LIN {X 0,Y 104.793,Z 356.414,A -85,B 0,C 180,E1 -28295.245,E2 -28295.245} C_VEL
LIN {X 0,Y 103.647,Z 359.104,A -85,B 0,C 180,E1 -28297.183,E2 -28297.183} C_VEL
LIN {X 0,Y 96.406,Z 367.355,A -85,B 0,C 180,E1 -28301.678,E2 -28301.678} C_VEL
LIN {X 0,Y 90.767,Z 372.964,A -85,B 0,C 180,E1 -28305.825,E2 -28305.825} C_VEL
LIN {X 0,Y 84.492,Z 378.456,A -85,B 0,C 180,E1 -28311.403,E2 -28311.403} C_VEL
LIN {X 0,Y 79.25,Z 382.759,A -85,B 0,C 180,E1 -28317.854,E2 -28317.854} C_VEL
LIN {X 0,Y 76.317,Z 385.034,A -85,B 0,C 180,E1 -28322.584,E2 -28322.584} C_VEL
LIN {X 0,Y 73.868,Z 386.882,A -85,B 0,C 180,E1 -28327.631,E2 -28327.631} C_VEL
LIN {X 0,Y 72.01,Z 388.266,A -85,B 0,C 180,E1 -28332.975,E2 -28332.975} C_VEL
LIN {X 0,Y 70.538,Z 389.359,A -85,B 0,C 180,E1 -28339.552,E2 -28339.552} C_VEL
LIN {X 0,Y 69.778,Z 389.739,A -85,B 0,C 180,E1 -28342.701,E2 -28342.701} C_VEL
LIN {X 0,Y 68.056,Z 390.083,A -85,B 0,C 180,E1 -28347.417,E2 -28347.417} C_VEL
LIN {X 0,Y 64.284,Z 389.837,A -85,B 0,C 180,E1 -28359.106,E2 -28359.106} C_VEL
LIN {X 0,Y 64.171,Z 389.276,A -85,B 0,C 180,E1 -28364.414,E2 -28364.414} C_VEL
LIN {X 0,Y 64.494,Z 388.958,A -85,B 0,C 180,E1 -28366.15,E2 -28366.15} C_VEL
LIN {X 0,Y 67.351,Z 387.167,A -85,B 0,C 180,E1 -28374.671,E2 -28374.671} C_VEL
LIN {X 0,Y 71.592,Z 384.296,A -85,B 0,C 180,E1 -28382.679,E2 -28382.679} C_VEL
LIN {X 0,Y 76.945,Z 380.402,A -85,B 0,C 180,E1 -28389.746,E2 -28389.746} C_VEL
LIN {X 0,Y 83.424,Z 375.369,A -85,B 0,C 180,E1 -28395.733,E2 -28395.733} C_VEL
LIN {X 0,Y 90.542,Z 369.031,A -85,B 0,C 180,E1 -28400.916,E2 -28400.916} C_VEL
LIN {X 0,Y 98.216,Z 361.109,A -85,B 0,C 180,E1 -28405.373,E2 -28405.373} C_VEL
LIN {X 0,Y 99.699,Z 358.129,A -85,B 0,C 180,E1 -28407.77,E2 -28407.77} C_VEL
LIN {X 0,Y 100.292,Z 356.377,A -85,B 0,C 180,E1 -28409.361,E2 -28409.361} C_VEL
LIN {X 0,Y 100.745,Z 353.085,A -85,B 0,C 180,E1 -28413.037,E2 -28413.037} C_VEL
LIN {X 0,Y 100.845,Z 351.331,A -85,B 0,C 180,E1 -28415.282,E2 -28415.282} C_VEL
LIN {X 0,Y 100.69,Z 348.475,A -85,B 0,C 180,E1 -28419.574,E2 -28419.574} C_VEL
LIN {X 0,Y 100.47,Z 346.218,A -85,B 0,C 180,E1 -28423.751,E2 -28423.751} C_VEL
LIN {X 0,Y 100.246,Z 344.108,A -85,B 0,C 180,E1 -28428.967,E2 -28428.967} C_VEL
LIN {X 0,Y 100.132,Z 342.512,A -85,B 0,C 180,E1 -28435.975,E2 -28435.975} C_VEL
LIN {X 0,Y 100.538,Z 341.834,A -85,B 0,C 180,E1 -28440,E2 -28440} C_VEL
LIN {X 0,Y 100.479,Z 343.621,A -85,B 0,C 180,E1 -28448.041,E2 -28448.041} C_VEL
LIN {X 0,Y 100.756,Z 345.239,A -85,B 0,C 180,E1 -28452.434,E2 -28452.434} C_VEL
LIN {X 0,Y 100.752,Z 348.841,A -85,B 0,C 180,E1 -28458.294,E2 -28458.294} C_VEL
LIN {X 0,Y 100.473,Z 352.18,A -85,B 0,C 180,E1 -28462.454,E2 -28462.454} C_VEL
LIN {X 0,Y 99.589,Z 357.923,A -85,B 0,C 180,E1 -28468.447,E2 -28468.447} C_VEL
LIN {X 0,Y 99.259,Z 359.239,A -85,B 0,C 180,E1 -28469.711,E2 -28469.711} C_VEL
LIN {X 0,Y 95.481,Z 365.627,A -85,B 0,C 180,E1 -28474.098,E2 -28474.098} C_VEL
LIN {X 0,Y 94.457,Z 367.013,A -85,B 0,C 180,E1 -28475.07,E2 -28475.07} C_VEL
LIN {X 0,Y 86.861,Z 374.432,A -85,B 0,C 180,E1 -28479.766,E2 -28479.766} C_VEL
LIN {X 0,Y 80.095,Z 380.399,A -85,B 0,C 180,E1 -28485.414,E2 -28485.414} C_VEL
LIN {X 0,Y 73.98,Z 385.109,A -85,B 0,C 180,E1 -28491.866,E2 -28491.866} C_VEL
LIN {X 0,Y 68.92,Z 388.71,A -85,B 0,C 180,E1 -28499.344,E2 -28499.344} C_VEL
LIN {X 0,Y 66.352,Z 390.571,A -85,B 0,C 180,E1 -28504.932,E2 -28504.932} C_VEL
LIN {X 0,Y 64.453,Z 391.97,A -85,B 0,C 180,E1 -28510.905,E2 -28510.905} C_VEL
LIN {X 0,Y 63.178,Z 392.971,A -85,B 0,C 180,E1 -28517.144,E2 -28517.144} C_VEL
LIN {X 0,Y 62.555,Z 393.585,A -85,B 0,C 180,E1 -28523.549,E2 -28523.549} C_VEL
LIN {X 0,Y 62.607,Z 393.802,A -85,B 0,C 180,E1 -28529.999,E2 -28529.999} C_VEL
LIN {X 0,Y 62.554,Z 393.565,A -85,B 0,C 180,E1 -28536.45,E2 -28536.45} C_VEL
LIN {X 0,Y 63.173,Z 392.94,A -85,B 0,C 180,E1 -28542.855,E2 -28542.855} C_VEL
LIN {X 0,Y 64.448,Z 391.926,A -85,B 0,C 180,E1 -28549.095,E2 -28549.095} C_VEL
LIN {X 0,Y 66.351,Z 390.508,A -85,B 0,C 180,E1 -28555.067,E2 -28555.067} C_VEL
LIN {X 0,Y 70.489,Z 387.549,A -85,B 0,C 180,E1 -28563.255,E2 -28563.255} C_VEL
LIN {X 0,Y 75.858,Z 383.553,A -85,B 0,C 180,E1 -28570.43,E2 -28570.43} C_VEL
LIN {X 0,Y 82.788,Z 377.962,A -85,B 0,C 180,E1 -28576.999,E2 -28576.999} C_VEL
LIN {X 0,Y 90.604,Z 370.717,A -85,B 0,C 180,E1 -28582.662,E2 -28582.662} C_VEL
LIN {X 0,Y 94.437,Z 366.784,A -85,B 0,C 180,E1 -28584.946,E2 -28584.946} C_VEL
LIN {X 0,Y 98.282,Z 360.732,A -85,B 0,C 180,E1 -28589.104,E2 -28589.104} C_VEL
LIN {X 0,Y 99.138,Z 359.09,A -85,B 0,C 180,E1 -28590.249,E2 -28590.249} C_VEL
LIN {X 0,Y 100.072,Z 354.239,A -85,B 0,C 180,E1 -28595.079,E2 -28595.079} C_VEL
LIN {X 0,Y 100.485,Z 350.318,A -85,B 0,C 180,E1 -28599.531,E2 -28599.531} C_VEL
LIN {X 0,Y 100.597,Z 347.225,A -85,B 0,C 180,E1 -28603.773,E2 -28603.773} C_VEL
LIN {X 0,Y 100.675,Z 345.864,A -85,B 0,C 180,E1 -28605.858,E2 -28605.858} C_VEL
LIN {X 0,Y 100.584,Z 344.822,A -85,B 0,C 180,E1 -28608.014,E2 -28608.014} C_VEL
LIN {X 0,Y 100.327,Z 343.386,A -85,B 0,C 180,E1 -28611.946,E2 -28611.946} C_VEL
LIN {X 0,Y 100.495,Z 341.438,A -85,B 0,C 180,E1 -28620,E2 -28620} C_VEL
LIN {X 0,Y 100.058,Z 343.703,A -85,B 0,C 180,E1 -28630.472,E2 -28630.472} C_VEL
LIN {X 0,Y 100.312,Z 345.977,A -85,B 0,C 180,E1 -28636.275,E2 -28636.275} C_VEL
LIN {X 0,Y 100.573,Z 349.257,A -85,B 0,C 180,E1 -28642.047,E2 -28642.047} C_VEL
LIN {X 0,Y 100.754,Z 351.181,A -85,B 0,C 180,E1 -28644.933,E2 -28644.933} C_VEL
LIN {X 0,Y 100.621,Z 353.725,A -85,B 0,C 180,E1 -28648.128,E2 -28648.128} C_VEL
LIN {X 0,Y 100.212,Z 356.032,A -85,B 0,C 180,E1 -28650.563,E2 -28650.563} C_VEL
LIN {X 0,Y 99.055,Z 359.33,A -85,B 0,C 180,E1 -28653.525,E2 -28653.525} C_VEL
LIN {X 0,Y 98.237,Z 360.784,A -85,B 0,C 180,E1 -28654.645,E2 -28654.645} C_VEL
LIN {X 0,Y 90.606,Z 368.761,A -85,B 0,C 180,E1 -28659.135,E2 -28659.135} C_VEL
LIN {X 0,Y 83.478,Z 375.163,A -85,B 0,C 180,E1 -28664.307,E2 -28664.307} C_VEL
LIN {X 0,Y 76.994,Z 380.242,A -85,B 0,C 180,E1 -28670.286,E2 -28670.286} C_VEL
LIN {X 0,Y 71.622,Z 384.178,A -85,B 0,C 180,E1 -28677.338,E2 -28677.338} C_VEL
LIN {X 0,Y 67.358,Z 387.082,A -85,B 0,C 180,E1 -28685.333,E2 -28685.333} C_VEL
LIN {X 0,Y 65.247,Z 388.467,A -85,B 0,C 180,E1 -28691.148,E2 -28691.148} C_VEL
LIN {X 0,Y 62.941,Z 390.052,A -85,B 0,C 180,E1 -28703.59,E2 -28703.59} C_VEL
LIN {X 0,Y 62.722,Z 390.274,A -85,B 0,C 180,E1 -28710.001,E2 -28710.001} C_VEL
LIN {X 0,Y 62.941,Z 390.078,A -85,B 0,C 180,E1 -28716.412,E2 -28716.412} C_VEL
LIN {X 0,Y 64.494,Z 388.958,A -85,B 0,C 180,E1 -28726.15,E2 -28726.15} C_VEL
LIN {X 0,Y 65.325,Z 388.093,A -85,B 0,C 180,E1 -28731.256,E2 -28731.256} C_VEL
LIN {X 0,Y 65.947,Z 386.149,A -85,B 0,C 180,E1 -28739.749,E2 -28739.749} C_VEL
LIN {X 0,Y 67.198,Z 384.11,A -85,B 0,C 180,E1 -28746.298,E2 -28746.298} C_VEL
LIN {X 0,Y 69.308,Z 382.218,A -85,B 0,C 180,E1 -28750.671,E2 -28750.671} C_VEL
LIN {X 0,Y 70.305,Z 381.487,A -85,B 0,C 180,E1 -28751.943,E2 -28751.943} C_VEL
LIN {X 0,Y 78.633,Z 375.567,A -85,B 0,C 180,E1 -28759.439,E2 -28759.439} C_VEL
LIN {X 0,Y 86.244,Z 369.229,A -85,B 0,C 180,E1 -28764.579,E2 -28764.579} C_VEL
LIN {X 0,Y 93.006,Z 362.777,A -85,B 0,C 180,E1 -28768.22,E2 -28768.22} C_VEL
LIN {X 0,Y 93.91,Z 361.331,A -85,B 0,C 180,E1 -28769.385,E2 -28769.385} C_VEL
LIN {X 0,Y 94.71,Z 359.575,A -85,B 0,C 180,E1 -28771.164,E2 -28771.164} C_VEL
LIN {X 0,Y 95.354,Z 356.566,A -85,B 0,C 180,E1 -28774.987,E2 -28774.987} C_VEL
LIN {X 0,Y 95.522,Z 354.36,A -85,B 0,C 180,E1 -28778.415,E2 -28778.415} C_VEL
LIN {X 0,Y 95.604,Z 351.962,A -85,B 0,C 180,E1 -28782.899,E2 -28782.899} C_VEL
LIN {X 0,Y 95.525,Z 350.184,A -85,B 0,C 180,E1 -28787.249,E2 -28787.249} C_VEL
LIN {X 0,Y 95.559,Z 348.88,A -85,B 0,C 180,E1 -28791.541,E2 -28791.541} C_VEL
LIN {X 0,Y 96.103,Z 347.425,A -85,B 0,C 180,E1 -28800,E2 -28800} C_VEL
LIN {X 0,Y 95.893,Z 349.285,A -85,B 0,C 180,E1 -28808.429,E2 -28808.429} C_VEL
LIN {X 0,Y 95.97,Z 350.846,A -85,B 0,C 180,E1 -28812.691,E2 -28812.691} C_VEL
LIN {X 0,Y 95.697,Z 353.545,A -85,B 0,C 180,E1 -28817.306,E2 -28817.306} C_VEL
LIN {X 0,Y 94.847,Z 357.84,A -85,B 0,C 180,E1 -28822.935,E2 -28822.935} C_VEL
LIN {X 0,Y 93.979,Z 361.101,A -85,B 0,C 180,E1 -28826.66,E2 -28826.66} C_VEL
LIN {X 0,Y 93.253,Z 362.663,A -85,B 0,C 180,E1 -28828.099,E2 -28828.099} C_VEL
LIN {X 0,Y 90.33,Z 366.803,A -85,B 0,C 180,E1 -28831.147,E2 -28831.147} C_VEL
LIN {X 0,Y 89.184,Z 368.175,A -85,B 0,C 180,E1 -28832.097,E2 -28832.097} C_VEL
LIN {X 0,Y 81.199,Z 375.347,A -85,B 0,C 180,E1 -28836.81,E2 -28836.81} C_VEL
LIN {X 0,Y 72.857,Z 381.889,A -85,B 0,C 180,E1 -28843.657,E2 -28843.657} C_VEL
LIN {X 0,Y 66.526,Z 386.217,A -85,B 0,C 180,E1 -28850.664,E2 -28850.664} C_VEL
LIN {X 0,Y 62.902,Z 388.511,A -85,B 0,C 180,E1 -28856.037,E2 -28856.037} C_VEL
LIN {X 0,Y 59.955,Z 390.37,A -85,B 0,C 180,E1 -28862.037,E2 -28862.037} C_VEL
LIN {X 0,Y 57.762,Z 391.77,A -85,B 0,C 180,E1 -28868.591,E2 -28868.591} C_VEL
LIN {X 0,Y 56.266,Z 392.772,A -85,B 0,C 180,E1 -28875.533,E2 -28875.533} C_VEL
LIN {X 0,Y 55.513,Z 393.385,A -85,B 0,C 180,E1 -28882.726,E2 -28882.726} C_VEL
LIN {X 0,Y 55.506,Z 393.602,A -85,B 0,C 180,E1 -28889.999,E2 -28889.999} C_VEL
LIN {X 0,Y 55.511,Z 393.366,A -85,B 0,C 180,E1 -28897.273,E2 -28897.273} C_VEL
LIN {X 0,Y 56.262,Z 392.74,A -85,B 0,C 180,E1 -28904.467,E2 -28904.467} C_VEL
LIN {X 0,Y 57.758,Z 391.725,A -85,B 0,C 180,E1 -28911.409,E2 -28911.409} C_VEL
LIN {X 0,Y 59.954,Z 390.306,A -85,B 0,C 180,E1 -28917.962,E2 -28917.962} C_VEL
LIN {X 0,Y 64.658,Z 387.348,A -85,B 0,C 180,E1 -28926.714,E2 -28926.714} C_VEL
LIN {X 0,Y 70.589,Z 383.351,A -85,B 0,C 180,E1 -28934.181,E2 -28934.181} C_VEL
LIN {X 0,Y 77.441,Z 378.285,A -85,B 0,C 180,E1 -28940.333,E2 -28940.333} C_VEL
LIN {X 0,Y 85.131,Z 371.751,A -85,B 0,C 180,E1 -28945.644,E2 -28945.644} C_VEL
LIN {X 0,Y 89.174,Z 367.943,A -85,B 0,C 180,E1 -28947.911,E2 -28947.911} C_VEL
LIN {X 0,Y 93.145,Z 362.521,A -85,B 0,C 180,E1 -28951.848,E2 -28951.848} C_VEL
LIN {X 0,Y 93.986,Z 360.476,A -85,B 0,C 180,E1 -28953.808,E2 -28953.808} C_VEL
LIN {X 0,Y 94.958,Z 356.609,A -85,B 0,C 180,E1 -28958.281,E2 -28958.281} C_VEL
LIN {X 0,Y 95.591,Z 353.198,A -85,B 0,C 180,E1 -28962.897,E2 -28962.897} C_VEL
LIN {X 0,Y 95.85,Z 350.624,A -85,B 0,C 180,E1 -28967.293,E2 -28967.293} C_VEL
LIN {X 0,Y 95.769,Z 349.057,A -85,B 0,C 180,E1 -28971.56,E2 -28971.56} C_VEL
LIN {X 0,Y 96.064,Z 347.06,A -85,B 0,C 180,E1 -28980,E2 -28980} C_VEL
LIN {X 0,Y 95.417,Z 348.65,A -85,B 0,C 180,E1 -28988.471,E2 -28988.471} C_VEL
LIN {X 0,Y 95.402,Z 349.929,A -85,B 0,C 180,E1 -28992.768,E2 -28992.768} C_VEL
LIN {X 0,Y 95.48,Z 351.717,A -85,B 0,C 180,E1 -28997.123,E2 -28997.123} C_VEL
LIN {X 0,Y 95.418,Z 355.078,A -85,B 0,C 180,E1 -29003.236,E2 -29003.236} C_VEL
LIN {X 0,Y 94.965,Z 358.049,A -85,B 0,C 180,E1 -29007.368,E2 -29007.368} C_VEL
LIN {X 0,Y 93.898,Z 361.013,A -85,B 0,C 180,E1 -29010.605,E2 -29010.605} C_VEL
LIN {X 0,Y 93.003,Z 362.465,A -85,B 0,C 180,E1 -29011.778,E2 -29011.778} C_VEL
LIN {X 0,Y 85.01,Z 370.125,A -85,B 0,C 180,E1 -29016.288,E2 -29016.288} C_VEL
LIN {X 0,Y 76.266,Z 377.17,A -85,B 0,C 180,E1 -29022.506,E2 -29022.506} C_VEL
LIN {X 0,Y 69.596,Z 381.857,A -85,B 0,C 180,E1 -29028.975,E2 -29028.975} C_VEL
LIN {X 0,Y 64.014,Z 385.437,A -85,B 0,C 180,E1 -29036.706,E2 -29036.706} C_VEL
LIN {X 0,Y 60.985,Z 387.283,A -85,B 0,C 180,E1 -29042.551,E2 -29042.551} C_VEL
LIN {X 0,Y 58.577,Z 388.667,A -85,B 0,C 180,E1 -29048.904,E2 -29048.904} C_VEL
LIN {X 0,Y 55.909,Z 390.252,A -85,B 0,C 180,E1 -29062.779,E2 -29062.779} C_VEL
LIN {X 0,Y 55.649,Z 390.474,A -85,B 0,C 180,E1 -29070.001,E2 -29070.001} C_VEL
LIN {X 0,Y 55.909,Z 390.277,A -85,B 0,C 180,E1 -29077.222,E2 -29077.222} C_VEL
LIN {X 0,Y 58.576,Z 388.725,A -85,B 0,C 180,E1 -29091.098,E2 -29091.098} C_VEL
LIN {X 0,Y 60.977,Z 387.366,A -85,B 0,C 180,E1 -29097.454,E2 -29097.454} C_VEL
LIN {X 0,Y 65.724,Z 384.495,A -85,B 0,C 180,E1 -29106.025,E2 -29106.025} C_VEL
LIN {X 0,Y 70.305,Z 381.487,A -85,B 0,C 180,E1 -29111.943,E2 -29111.943} C_VEL
LIN {X 0,Y 73.125,Z 379.246,A -85,B 0,C 180,E1 -29115.692,E2 -29115.692} C_VEL
LIN {X 0,Y 76.946,Z 375.192,A -85,B 0,C 180,E1 -29121.978,E2 -29121.978} C_VEL
LIN {X 0,Y 81.339,Z 370.522,A -85,B 0,C 180,E1 -29127.46,E2 -29127.46} C_VEL
LIN {X 0,Y 84.847,Z 367.257,A -85,B 0,C 180,E1 -29129.866,E2 -29129.866} C_VEL
LIN {X 0,Y 88.03,Z 364.33,A -85,B 0,C 180,E1 -29131.428,E2 -29131.428} C_VEL
LIN {X 0,Y 88.837,Z 363.193,A -85,B 0,C 180,E1 -29132.531,E2 -29132.531} C_VEL
LIN {X 0,Y 89.409,Z 361.74,A -85,B 0,C 180,E1 -29134.408,E2 -29134.408} C_VEL
LIN {X 0,Y 89.91,Z 360.045,A -85,B 0,C 180,E1 -29136.993,E2 -29136.993} C_VEL
LIN {X 0,Y 90.324,Z 357.435,A -85,B 0,C 180,E1 -29141.866,E2 -29141.866} C_VEL
LIN {X 0,Y 90.45,Z 355.628,A -85,B 0,C 180,E1 -29146.52,E2 -29146.52} C_VEL
LIN {X 0,Y 90.604,Z 354.253,A -85,B 0,C 180,E1 -29151.075,E2 -29151.075} C_VEL
LIN {X 0,Y 91.347,Z 352.774,A -85,B 0,C 180,E1 -29160,E2 -29160} C_VEL
LIN {X 0,Y 91.033,Z 353.566,A -85,B 0,C 180,E1 -29164.428,E2 -29164.428} C_VEL
LIN {X 0,Y 90.954,Z 354.674,A -85,B 0,C 180,E1 -29168.89,E2 -29168.89} C_VEL
LIN {X 0,Y 90.738,Z 356.498,A -85,B 0,C 180,E1 -29173.436,E2 -29173.436} C_VEL
LIN {X 0,Y 90.028,Z 359.286,A -85,B 0,C 180,E1 -29178.195,E2 -29178.195} C_VEL
LIN {X 0,Y 88.752,Z 363.063,A -85,B 0,C 180,E1 -29183.324,E2 -29183.324} C_VEL
LIN {X 0,Y 88.142,Z 364.523,A -85,B 0,C 180,E1 -29185.06,E2 -29185.06} C_VEL
LIN {X 0,Y 85.452,Z 367.967,A -85,B 0,C 180,E1 -29187.853,E2 -29187.853} C_VEL
LIN {X 0,Y 82.726,Z 370.525,A -85,B 0,C 180,E1 -29189.448,E2 -29189.448} C_VEL
LIN {X 0,Y 75.787,Z 376.169,A -85,B 0,C 180,E1 -29193.424,E2 -29193.424} C_VEL
LIN {X 0,Y 68.138,Z 381.69,A -85,B 0,C 180,E1 -29199.323,E2 -29199.323} C_VEL
LIN {X 0,Y 61.187,Z 386.018,A -85,B 0,C 180,E1 -29206.435,E2 -29206.435} C_VEL
LIN {X 0,Y 57.141,Z 388.311,A -85,B 0,C 180,E1 -29212.049,E2 -29212.049} C_VEL
LIN {X 0,Y 53.751,Z 390.17,A -85,B 0,C 180,E1 -29218.465,E2 -29218.465} C_VEL
LIN {X 0,Y 51.175,Z 391.569,A -85,B 0,C 180,E1 -29225.669,E2 -29225.669} C_VEL
LIN {X 0,Y 48.473,Z 393.185,A -85,B 0,C 180,E1 -29241.663,E2 -29241.663} C_VEL
LIN {X 0,Y 48.423,Z 393.403,A -85,B 0,C 180,E1 -29249.999,E2 -29249.999} C_VEL
LIN {X 0,Y 48.472,Z 393.165,A -85,B 0,C 180,E1 -29258.336,E2 -29258.336} C_VEL
LIN {X 0,Y 51.171,Z 391.524,A -85,B 0,C 180,E1 -29274.332,E2 -29274.332} C_VEL
LIN {X 0,Y 53.749,Z 390.104,A -85,B 0,C 180,E1 -29281.535,E2 -29281.535} C_VEL
LIN {X 0,Y 59.088,Z 387.146,A -85,B 0,C 180,E1 -29290.856,E2 -29290.856} C_VEL
LIN {X 0,Y 65.674,Z 383.15,A -85,B 0,C 180,E1 -29298.511,E2 -29298.511} C_VEL
LIN {X 0,Y 73.697,Z 377.617,A -85,B 0,C 180,E1 -29305.098,E2 -29305.098} C_VEL
LIN {X 0,Y 82.733,Z 370.311,A -85,B 0,C 180,E1 -29310.542,E2 -29310.542} C_VEL
LIN {X 0,Y 84.169,Z 369.074,A -85,B 0,C 180,E1 -29311.25,E2 -29311.25} C_VEL
LIN {X 0,Y 86.559,Z 366.349,A -85,B 0,C 180,E1 -29313.268,E2 -29313.268} C_VEL
LIN {X 0,Y 88.046,Z 364.33,A -85,B 0,C 180,E1 -29314.946,E2 -29314.946} C_VEL
LIN {X 0,Y 89.419,Z 360.838,A -85,B 0,C 180,E1 -29319.29,E2 -29319.29} C_VEL
LIN {X 0,Y 90.216,Z 358.113,A -85,B 0,C 180,E1 -29323.296,E2 -29323.296} C_VEL
LIN {X 0,Y 90.659,Z 356.253,A -85,B 0,C 180,E1 -29326.552,E2 -29326.552} C_VEL
LIN {X 0,Y 90.83,Z 354.468,A -85,B 0,C 180,E1 -29331.098,E2 -29331.098} C_VEL
LIN {X 0,Y 91.322,Z 352.439,A -85,B 0,C 180,E1 -29340,E2 -29340} C_VEL
LIN {X 0,Y 90.492,Z 354.013,A -85,B 0,C 180,E1 -29348.936,E2 -29348.936} C_VEL
LIN {X 0,Y 90.342,Z 355.38,A -85,B 0,C 180,E1 -29353.496,E2 -29353.496} C_VEL
LIN {X 0,Y 90.19,Z 357.231,A -85,B 0,C 180,E1 -29358.162,E2 -29358.162} C_VEL
LIN {X 0,Y 89.854,Z 359.785,A -85,B 0,C 180,E1 -29363.022,E2 -29363.022} C_VEL
LIN {X 0,Y 89.401,Z 361.434,A -85,B 0,C 180,E1 -29365.592,E2 -29365.592} C_VEL
LIN {X 0,Y 88.812,Z 362.868,A -85,B 0,C 180,E1 -29367.39,E2 -29367.39} C_VEL
LIN {X 0,Y 87.752,Z 364.313,A -85,B 0,C 180,E1 -29368.721,E2 -29368.721} C_VEL
LIN {X 0,Y 79.645,Z 371.436,A -85,B 0,C 180,E1 -29373.04,E2 -29373.04} C_VEL
LIN {X 0,Y 71.657,Z 377.371,A -85,B 0,C 180,E1 -29378.314,E2 -29378.314} C_VEL
LIN {X 0,Y 64.397,Z 382.058,A -85,B 0,C 180,E1 -29384.816,E2 -29384.816} C_VEL
LIN {X 0,Y 58.204,Z 385.638,A -85,B 0,C 180,E1 -29392.862,E2 -29392.862} C_VEL
LIN {X 0,Y 54.766,Z 387.484,A -85,B 0,C 180,E1 -29399.116,E2 -29399.116} C_VEL
LIN {X 0,Y 50.039,Z 389.85,A -85,B 0,C 180,E1 -29413.687,E2 -29413.687} C_VEL
LIN {X 0,Y 48.875,Z 390.452,A -85,B 0,C 180,E1 -29421.733,E2 -29421.733} C_VEL
LIN {X 0,Y 48.564,Z 390.673,A -85,B 0,C 180,E1 -29430.001,E2 -29430.001} C_VEL
LIN {X 0,Y 48.875,Z 390.477,A -85,B 0,C 180,E1 -29438.268,E2 -29438.268} C_VEL
LIN {X 0,Y 50.039,Z 389.891,A -85,B 0,C 180,E1 -29446.315,E2 -29446.315} C_VEL
LIN {X 0,Y 54.759,Z 387.566,A -85,B 0,C 180,E1 -29460.89,E2 -29460.89} C_VEL
LIN {X 0,Y 60.125,Z 384.694,A -85,B 0,C 180,E1 -29470.009,E2 -29470.009} C_VEL
LIN {X 0,Y 66.647,Z 380.799,A -85,B 0,C 180,E1 -29477.576,E2 -29477.576} C_VEL
LIN {X 0,Y 74.214,Z 375.766,A -85,B 0,C 180,E1 -29483.606,E2 -29483.606} C_VEL
LIN {X 0,Y 82.337,Z 369.426,A -85,B 0,C 180,E1 -29488.603,E2 -29488.603} C_VEL
LIN {X 0,Y 84.847,Z 367.257,A -85,B 0,C 180,E1 -29489.866,E2 -29489.866} C_VEL
LIN {X 0,Y 86.035,Z 365.951,A -85,B 0,C 180,E1 -29490.983,E2 -29490.983} C_VEL
LIN {X 0,Y 86.574,Z 364.684,A -85,B 0,C 180,E1 -29492.858,E2 -29492.858} C_VEL
LIN {X 0,Y 86.25,Z 363.534,A -85,B 0,C 180,E1 -29495.807,E2 -29495.807} C_VEL
LIN {X 0,Y 84.738,Z 361.87,A -85,B 0,C 180,E1 -29502.763,E2 -29502.763} C_VEL
LIN {X 0,Y 84.775,Z 361.518,A -85,B 0,C 180,E1 -29503.757,E2 -29503.757} C_VEL
LIN {X 0,Y 85.002,Z 360.784,A -85,B 0,C 180,E1 -29505.638,E2 -29505.638} C_VEL
LIN {X 0,Y 85.387,Z 359.235,A -85,B 0,C 180,E1 -29511.007,E2 -29511.007} C_VEL
LIN {X 0,Y 86.258,Z 357.827,A -85,B 0,C 180,E1 -29520,E2 -29520} C_VEL
LIN {X 0,Y 85.893,Z 358.627,A -85,B 0,C 180,E1 -29524.693,E2 -29524.693} C_VEL
LIN {X 0,Y 85.586,Z 360.011,A -85,B 0,C 180,E1 -29529.801,E2 -29529.801} C_VEL
LIN {X 0,Y 85.054,Z 361.912,A -85,B 0,C 180,E1 -29534.352,E2 -29534.352} C_VEL
LIN {X 0,Y 83.76,Z 365.052,A -85,B 0,C 180,E1 -29539.61,E2 -29539.61} C_VEL
LIN {X 0,Y 83.086,Z 366.35,A -85,B 0,C 180,E1 -29541.492,E2 -29541.492} C_VEL
LIN {X 0,Y 82.111,Z 367.751,A -85,B 0,C 180,E1 -29543.057,E2 -29543.057} C_VEL
LIN {X 0,Y 80.884,Z 369.083,A -85,B 0,C 180,E1 -29544.166,E2 -29544.166} C_VEL
LIN {X 0,Y 72.097,Z 375.97,A -85,B 0,C 180,E1 -29548.677,E2 -29548.677} C_VEL
LIN {X 0,Y 63.861,Z 381.491,A -85,B 0,C 180,E1 -29554.371,E2 -29554.371} C_VEL
LIN {X 0,Y 56.23,Z 385.818,A -85,B 0,C 180,E1 -29561.415,E2 -29561.415} C_VEL
LIN {X 0,Y 51.718,Z 388.112,A -85,B 0,C 180,E1 -29567.197,E2 -29567.197} C_VEL
LIN {X 0,Y 47.811,Z 389.969,A -85,B 0,C 180,E1 -29573.985,E2 -29573.985} C_VEL
LIN {X 0,Y 42.608,Z 392.371,A -85,B 0,C 180,E1 -29590.737,E2 -29590.737} C_VEL
LIN {X 0,Y 41.447,Z 392.985,A -85,B 0,C 180,E1 -29600.236,E2 -29600.236} C_VEL
LIN {X 0,Y 41.322,Z 393.203,A -85,B 0,C 180,E1 -29609.999,E2 -29609.999} C_VEL
LIN {X 0,Y 41.445,Z 392.965,A -85,B 0,C 180,E1 -29619.762,E2 -29619.762} C_VEL
LIN {X 0,Y 44.764,Z 391.322,A -85,B 0,C 180,E1 -29638.098,E2 -29638.098} C_VEL
LIN {X 0,Y 47.809,Z 389.903,A -85,B 0,C 180,E1 -29646.014,E2 -29646.014} C_VEL
LIN {X 0,Y 53.897,Z 386.944,A -85,B 0,C 180,E1 -29655.821,E2 -29655.821} C_VEL
LIN {X 0,Y 61.195,Z 382.949,A -85,B 0,C 180,E1 -29663.505,E2 -29663.505} C_VEL
LIN {X 0,Y 69.889,Z 377.394,A -85,B 0,C 180,E1 -29669.921,E2 -29669.921} C_VEL
LIN {X 0,Y 79.473,Z 370.109,A -85,B 0,C 180,E1 -29675.016,E2 -29675.016} C_VEL
LIN {X 0,Y 80.866,Z 368.863,A -85,B 0,C 180,E1 -29675.859,E2 -29675.859} C_VEL
LIN {X 0,Y 82.087,Z 367.508,A -85,B 0,C 180,E1 -29676.98,E2 -29676.98} C_VEL
LIN {X 0,Y 83.037,Z 366.104,A -85,B 0,C 180,E1 -29678.592,E2 -29678.592} C_VEL
LIN {X 0,Y 84.421,Z 363.126,A -85,B 0,C 180,E1 -29683.06,E2 -29683.06} C_VEL
LIN {X 0,Y 85.379,Z 360.52,A -85,B 0,C 180,E1 -29688.127,E2 -29688.127} C_VEL
LIN {X 0,Y 85.536,Z 359.659,A -85,B 0,C 180,E1 -29690.542,E2 -29690.542} C_VEL
LIN {X 0,Y 85.776,Z 358.427,A -85,B 0,C 180,E1 -29695.3,E2 -29695.3} C_VEL
LIN {X 0,Y 86.238,Z 357.532,A -85,B 0,C 180,E1 -29700,E2 -29700} C_VEL
LIN {X 0,Y 85.231,Z 359.144,A -85,B 0,C 180,E1 -29709.493,E2 -29709.493} C_VEL
LIN {X 0,Y 84.893,Z 360.579,A -85,B 0,C 180,E1 -29714.381,E2 -29714.381} C_VEL
LIN {X 0,Y 84.51,Z 362.522,A -85,B 0,C 180,E1 -29719.43,E2 -29719.43} C_VEL
LIN {X 0,Y 83.936,Z 364.311,A -85,B 0,C 180,E1 -29722.923,E2 -29722.923} C_VEL
LIN {X 0,Y 83.305,Z 365.61,A -85,B 0,C 180,E1 -29724.95,E2 -29724.95} C_VEL
LIN {X 0,Y 74.579,Z 372.746,A -85,B 0,C 180,E1 -29729.347,E2 -29729.347} C_VEL
LIN {X 0,Y 67.485,Z 377.573,A -85,B 0,C 180,E1 -29733.579,E2 -29733.579} C_VEL
LIN {X 0,Y 59.601,Z 382.259,A -85,B 0,C 180,E1 -29739.963,E2 -29739.963} C_VEL
LIN {X 0,Y 52.718,Z 385.838,A -85,B 0,C 180,E1 -29748.199,E2 -29748.199} C_VEL
LIN {X 0,Y 48.802,Z 387.684,A -85,B 0,C 180,E1 -29754.828,E2 -29754.828} C_VEL
LIN {X 0,Y 43.275,Z 390.05,A -85,B 0,C 180,E1 -29771.047,E2 -29771.047} C_VEL
LIN {X 0,Y 41.878,Z 390.651,A -85,B 0,C 180,E1 -29780.34,E2 -29780.34} C_VEL
LIN {X 0,Y 41.469,Z 390.873,A -85,B 0,C 180,E1 -29790.001,E2 -29790.001} C_VEL
LIN {X 0,Y 41.878,Z 390.676,A -85,B 0,C 180,E1 -29799.662,E2 -29799.662} C_VEL
LIN {X 0,Y 43.275,Z 390.091,A -85,B 0,C 180,E1 -29808.955,E2 -29808.955} C_VEL
LIN {X 0,Y 48.795,Z 387.765,A -85,B 0,C 180,E1 -29825.18,E2 -29825.18} C_VEL
LIN {X 0,Y 54.876,Z 384.894,A -85,B 0,C 180,E1 -29834.782,E2 -29834.782} C_VEL
LIN {X 0,Y 62.083,Z 380.998,A -85,B 0,C 180,E1 -29842.414,E2 -29842.414} C_VEL
LIN {X 0,Y 70.237,Z 375.964,A -85,B 0,C 180,E1 -29848.27,E2 -29848.27} C_VEL
LIN {X 0,Y 78.877,Z 369.624,A -85,B 0,C 180,E1 -29853.001,E2 -29853.001} C_VEL
LIN {X 0,Y 83.358,Z 365.849,A -85,B 0,C 180,E1 -29855.067,E2 -29855.067} C_VEL
LIN {X 0,Y 83.939,Z 364.592,A -85,B 0,C 180,E1 -29857.074,E2 -29857.074} C_VEL
LIN {X 0,Y 84.6,Z 362.746,A -85,B 0,C 180,E1 -29860.592,E2 -29860.592} C_VEL
LIN {X 0,Y 84.775,Z 361.518,A -85,B 0,C 180,E1 -29863.757,E2 -29863.757} C_VEL
LIN {X 0,Y 84.794,Z 360.762,A -85,B 0,C 180,E1 -29866.381,E2 -29866.381} C_VEL
LIN {X 0,Y 84.192,Z 360.424,A -85,B 0,C 180,E1 -29870.396,E2 -29870.396} C_VEL
LIN {X 0,Y 83.155,Z 360.805,A -85,B 0,C 180,E1 -29874.435,E2 -29874.435} C_VEL
LIN {X 0,Y 81.553,Z 362.054,A -85,B 0,C 180,E1 -29880.017,E2 -29880.017} C_VEL
LIN {X 0,Y 80.321,Z 363.638,A -85,B 0,C 180,E1 -29885.713,E2 -29885.713} C_VEL
LIN {X 0,Y 79.909,Z 364.849,A -85,B 0,C 180,E1 -29890.131,E2 -29890.131} C_VEL
LIN {X 0,Y 79.419,Z 366.008,A -85,B 0,C 180,E1 -29893.236,E2 -29893.236} C_VEL
LIN {X 0,Y 78.799,Z 367.154,A -85,B 0,C 180,E1 -29895.519,E2 -29895.519} C_VEL
LIN {X 0,Y 77.775,Z 368.861,A -85,B 0,C 180,E1 -29898.457,E2 -29898.457} C_VEL
LIN {X 0,Y 76.673,Z 370.131,A -85,B 0,C 180,E1 -29900.047,E2 -29900.047} C_VEL
LIN {X 0,Y 66.888,Z 377.161,A -85,B 0,C 180,E1 -29904.545,E2 -29904.545} C_VEL
LIN {X 0,Y 57.253,Z 382.877,A -85,B 0,C 180,E1 -29910.763,E2 -29910.763} C_VEL
LIN {X 0,Y 49.2,Z 386.838,A -85,B 0,C 180,E1 -29918.218,E2 -29918.218} C_VEL
LIN {X 0,Y 42.247,Z 389.769,A -85,B 0,C 180,E1 -29928.284,E2 -29928.284} C_VEL
LIN {X 0,Y 35.968,Z 392.171,A -85,B 0,C 180,E1 -29946.995,E2 -29946.995} C_VEL
LIN {X 0,Y 34.469,Z 392.786,A -85,B 0,C 180,E1 -29958.234,E2 -29958.234} C_VEL
LIN {X 0,Y 34.237,Z 393.004,A -85,B 0,C 180,E1 -29969.999,E2 -29969.999} C_VEL
LIN {X 0,Y 34.467,Z 392.765,A -85,B 0,C 180,E1 -29981.764,E2 -29981.764} C_VEL
LIN {X 0,Y 38.622,Z 391.121,A -85,B 0,C 180,E1 -30003.086,E2 -30003.086} C_VEL
LIN {X 0,Y 42.245,Z 389.701,A -85,B 0,C 180,E1 -30011.716,E2 -30011.716} C_VEL
LIN {X 0,Y 49.197,Z 386.743,A -85,B 0,C 180,E1 -30021.785,E2 -30021.785} C_VEL
LIN {X 0,Y 57.253,Z 382.747,A -85,B 0,C 180,E1 -30029.234,E2 -30029.234} C_VEL
LIN {X 0,Y 66.272,Z 377.416,A -85,B 0,C 180,E1 -30035.05,E2 -30035.05} C_VEL
LIN {X 0,Y 75.166,Z 371.144,A -85,B 0,C 180,E1 -30039.226,E2 -30039.226} C_VEL
LIN {X 0,Y 77.188,Z 369.352,A -85,B 0,C 180,E1 -30040.579,E2 -30040.579} C_VEL
LIN {X 0,Y 77.977,Z 368.283,A -85,B 0,C 180,E1 -30042.173,E2 -30042.173} C_VEL
LIN {X 0,Y 79.372,Z 365.753,A -85,B 0,C 180,E1 -30046.904,E2 -30046.904} C_VEL
LIN {X 0,Y 79.961,Z 364.545,A -85,B 0,C 180,E1 -30049.876,E2 -30049.876} C_VEL
LIN {X 0,Y 80.327,Z 363.25,A -85,B 0,C 180,E1 -30054.981,E2 -30054.981} C_VEL
LIN {X 0,Y 80.88,Z 362.323,A -85,B 0,C 180,E1 -30060,E2 -30060} C_VEL
LIN {X 0,Y 79.819,Z 363.489,A -85,B 0,C 180,E1 -30067.499,E2 -30067.499} C_VEL
LIN {X 0,Y 79.365,Z 364.731,A -85,B 0,C 180,E1 -30073.074,E2 -30073.074} C_VEL
LIN {X 0,Y 78.829,Z 366.402,A -85,B 0,C 180,E1 -30078.183,E2 -30078.183} C_VEL
LIN {X 0,Y 78.21,Z 367.693,A -85,B 0,C 180,E1 -30081.066,E2 -30081.066} C_VEL
LIN {X 0,Y 72.868,Z 371.84,A -85,B 0,C 180,E1 -30083.616,E2 -30083.616} C_VEL
LIN {X 0,Y 63.834,Z 377.774,A -85,B 0,C 180,E1 -30088.264,E2 -30088.264} C_VEL
LIN {X 0,Y 55.309,Z 382.46,A -85,B 0,C 180,E1 -30094.317,E2 -30094.317} C_VEL
LIN {X 0,Y 47.665,Z 386.039,A -85,B 0,C 180,E1 -30102.505,E2 -30102.505} C_VEL
LIN {X 0,Y 43.192,Z 387.885,A -85,B 0,C 180,E1 -30109.395,E2 -30109.395} C_VEL
LIN {X 0,Y 39.454,Z 389.268,A -85,B 0,C 180,E1 -30117.698,E2 -30117.698} C_VEL
LIN {X 0,Y 34.895,Z 390.851,A -85,B 0,C 180,E1 -30138.382,E2 -30138.382} C_VEL
LIN {X 0,Y 34.391,Z 391.072,A -85,B 0,C 180,E1 -30150.001,E2 -30150.001} C_VEL
LIN {X 0,Y 34.895,Z 390.876,A -85,B 0,C 180,E1 -30161.62,E2 -30161.62} C_VEL
LIN {X 0,Y 39.452,Z 389.323,A -85,B 0,C 180,E1 -30182.306,E2 -30182.306} C_VEL
LIN {X 0,Y 43.186,Z 387.965,A -85,B 0,C 180,E1 -30190.615,E2 -30190.615} C_VEL
LIN {X 0,Y 50.069,Z 385.093,A -85,B 0,C 180,E1 -30200.536,E2 -30200.536} C_VEL
LIN {X 0,Y 58.031,Z 381.196,A -85,B 0,C 180,E1 -30207.969,E2 -30207.969} C_VEL
LIN {X 0,Y 66.78,Z 376.162,A -85,B 0,C 180,E1 -30213.453,E2 -30213.453} C_VEL
LIN {X 0,Y 75.924,Z 369.821,A -85,B 0,C 180,E1 -30217.77,E2 -30217.77} C_VEL
LIN {X 0,Y 78.224,Z 367.936,A -85,B 0,C 180,E1 -30218.937,E2 -30218.937} C_VEL
LIN {X 0,Y 78.914,Z 366.61,A -85,B 0,C 180,E1 -30221.838,E2 -30221.838} C_VEL
LIN {X 0,Y 79.46,Z 364.991,A -85,B 0,C 180,E1 -30226.638,E2 -30226.638} C_VEL
LIN {X 0,Y 79.743,Z 364.197,A -85,B 0,C 180,E1 -30229.847,E2 -30229.847} C_VEL
LIN {X 0,Y 80.241,Z 363.215,A -85,B 0,C 180,E1 -30234.975,E2 -30234.975} C_VEL
LIN {X 0,Y 80.915,Z 362.58,A -85,B 0,C 180,E1 -30240,E2 -30240} C_VEL
LIN {X 0,Y 80.321,Z 363.638,A -85,B 0,C 180,E1 -30245.713,E2 -30245.713} C_VEL
LIN {X 0,Y 79.4,Z 364.879,A -85,B 0,C 180,E1 -30248.439,E2 -30248.439} C_VEL
LIN {X 0,Y 77.728,Z 366.694,A -85,B 0,C 180,E1 -30250.87,E2 -30250.87} C_VEL
LIN {X 0,Y 74.664,Z 369.556,A -85,B 0,C 180,E1 -30253.688,E2 -30253.688} C_VEL
LIN {X 0,Y 70.87,Z 372.569,A -85,B 0,C 180,E1 -30256.009,E2 -30256.009} C_VEL
LIN {X 0,Y 68.742,Z 374.071,A -85,B 0,C 180,E1 -30256.918,E2 -30256.918} C_VEL
LIN {X 0,Y 60.111,Z 379.399,A -85,B 0,C 180,E1 -30260.714,E2 -30260.714} C_VEL
LIN {X 0,Y 50.925,Z 384.111,A -85,B 0,C 180,E1 -30266.227,E2 -30266.227} C_VEL
LIN {X 0,Y 42.37,Z 387.712,A -85,B 0,C 180,E1 -30273.966,E2 -30273.966} C_VEL
LIN {X 0,Y 37.224,Z 389.569,A -85,B 0,C 180,E1 -30280.954,E2 -30280.954} C_VEL
LIN {X 0,Y 32.888,Z 390.968,A -85,B 0,C 180,E1 -30290.126,E2 -30290.126} C_VEL
LIN {X 0,Y 27.538,Z 392.586,A -85,B 0,C 180,E1 -30315.212,E2 -30315.212} C_VEL
LIN {X 0,Y 27.123,Z 392.803,A -85,B 0,C 180,E1 -30329.999,E2 -30329.999} C_VEL
LIN {X 0,Y 27.537,Z 392.564,A -85,B 0,C 180,E1 -30344.785,E2 -30344.785} C_VEL
LIN {X 0,Y 32.886,Z 390.92,A -85,B 0,C 180,E1 -30369.875,E2 -30369.875} C_VEL
LIN {X 0,Y 37.222,Z 389.5,A -85,B 0,C 180,E1 -30379.047,E2 -30379.047} C_VEL
LIN {X 0,Y 45.136,Z 386.541,A -85,B 0,C 180,E1 -30388.912,E2 -30388.912} C_VEL
LIN {X 0,Y 53.962,Z 382.546,A -85,B 0,C 180,E1 -30395.737,E2 -30395.737} C_VEL
LIN {X 0,Y 64.857,Z 376.403,A -85,B 0,C 180,E1 -30401.465,E2 -30401.465} C_VEL
LIN {X 0,Y 71.307,Z 372.113,A -85,B 0,C 180,E1 -30403.935,E2 -30403.935} C_VEL
LIN {X 0,Y 72.648,Z 370.909,A -85,B 0,C 180,E1 -30405.33,E2 -30405.33} C_VEL
LIN {X 0,Y 73.799,Z 369.266,A -85,B 0,C 180,E1 -30409.02,E2 -30409.02} C_VEL
LIN {X 0,Y 74.603,Z 367.776,A -85,B 0,C 180,E1 -30414.595,E2 -30414.595} C_VEL
LIN {X 0,Y 75.257,Z 366.822,A -85,B 0,C 180,E1 -30420,E2 -30420} C_VEL
LIN {X 0,Y 74.154,Z 367.802,A -85,B 0,C 180,E1 -30427.055,E2 -30427.055} C_VEL
LIN {X 0,Y 73.775,Z 368.484,A -85,B 0,C 180,E1 -30430.984,E2 -30430.984} C_VEL
LIN {X 0,Y 72.996,Z 370.063,A -85,B 0,C 180,E1 -30436.789,E2 -30436.789} C_VEL
LIN {X 0,Y 68.739,Z 373.149,A -85,B 0,C 180,E1 -30438.962,E2 -30438.962} C_VEL
LIN {X 0,Y 60.798,Z 377.975,A -85,B 0,C 180,E1 -30442.367,E2 -30442.367} C_VEL
LIN {X 0,Y 51.643,Z 382.661,A -85,B 0,C 180,E1 -30447.802,E2 -30447.802} C_VEL
LIN {X 0,Y 43.192,Z 386.239,A -85,B 0,C 180,E1 -30455.555,E2 -30455.555} C_VEL
LIN {X 0,Y 38.088,Z 388.085,A -85,B 0,C 180,E1 -30462.434,E2 -30462.434} C_VEL
LIN {X 0,Y 30.201,Z 390.451,A -85,B 0,C 180,E1 -30482.264,E2 -30482.264} C_VEL
LIN {X 0,Y 27.972,Z 391.052,A -85,B 0,C 180,E1 -30495.45,E2 -30495.45} C_VEL
LIN {X 0,Y 27.295,Z 391.272,A -85,B 0,C 180,E1 -30510.001,E2 -30510.001} C_VEL
LIN {X 0,Y 27.973,Z 391.076,A -85,B 0,C 180,E1 -30524.553,E2 -30524.553} C_VEL
LIN {X 0,Y 30.201,Z 390.49,A -85,B 0,C 180,E1 -30537.739,E2 -30537.739} C_VEL
LIN {X 0,Y 38.082,Z 388.164,A -85,B 0,C 180,E1 -30557.579,E2 -30557.579} C_VEL
LIN {X 0,Y 45.875,Z 385.293,A -85,B 0,C 180,E1 -30567.417,E2 -30567.417} C_VEL
LIN {X 0,Y 54.604,Z 381.394,A -85,B 0,C 180,E1 -30574.286,E2 -30574.286} C_VEL
LIN {X 0,Y 63.925,Z 376.36,A -85,B 0,C 180,E1 -30579.149,E2 -30579.149} C_VEL
LIN {X 0,Y 71.857,Z 371.19,A -85,B 0,C 180,E1 -30582.351,E2 -30582.351} C_VEL
LIN {X 0,Y 73.085,Z 370.243,A -85,B 0,C 180,E1 -30583.232,E2 -30583.232} C_VEL
LIN {X 0,Y 73.866,Z 368.664,A -85,B 0,C 180,E1 -30589.03,E2 -30589.03} C_VEL
LIN {X 0,Y 74.501,Z 367.702,A -85,B 0,C 180,E1 -30594.587,E2 -30594.587} C_VEL
LIN {X 0,Y 75.306,Z 367.045,A -85,B 0,C 180,E1 -30600,E2 -30600} C_VEL
LIN {X 0,Y 74.65,Z 367.987,A -85,B 0,C 180,E1 -30605.402,E2 -30605.402} C_VEL
LIN {X 0,Y 73.835,Z 369.47,A -85,B 0,C 180,E1 -30610.974,E2 -30610.974} C_VEL
LIN {X 0,Y 72.653,Z 371.135,A -85,B 0,C 180,E1 -30614.68,E2 -30614.68} C_VEL
LIN {X 0,Y 71.298,Z 372.316,A -85,B 0,C 180,E1 -30616.035,E2 -30616.035} C_VEL
LIN {X 0,Y 68.742,Z 374.071,A -85,B 0,C 180,E1 -30616.918,E2 -30616.918} C_VEL
LIN {X 0,Y 63.873,Z 377.085,A -85,B 0,C 180,E1 -30618.208,E2 -30618.208} C_VEL
LIN {X 0,Y 55.016,Z 381.427,A -85,B 0,C 180,E1 -30619.289,E2 -30619.289} C_VEL
LIN {X 0,Y 45.867,Z 385.027,A -85,B 0,C 180,E1 -30620.928,E2 -30620.928} C_VEL
LIN {X 0,Y 40.64,Z 386.879,A -85,B 0,C 180,E1 -30623.695,E2 -30623.695} C_VEL
LIN {X 0,Y 32.989,Z 389.369,A -85,B 0,C 180,E1 -30631.55,E2 -30631.55} C_VEL
LIN {X 0,Y 27.791,Z 390.768,A -85,B 0,C 180,E1 -30640.65,E2 -30640.65} C_VEL
LIN {X 0,Y 20.746,Z 392.386,A -85,B 0,C 180,E1 -30670.196,E2 -30670.196} C_VEL
LIN {X 0,Y 20.015,Z 392.603,A -85,B 0,C 180,E1 -30689.998,E2 -30689.998} C_VEL
LIN {X 0,Y 20.744,Z 392.364,A -85,B 0,C 180,E1 -30709.802,E2 -30709.802} C_VEL
LIN {X 0,Y 27.788,Z 390.719,A -85,B 0,C 180,E1 -30739.351,E2 -30739.351} C_VEL
LIN {X 0,Y 32.987,Z 389.298,A -85,B 0,C 180,E1 -30748.451,E2 -30748.451} C_VEL
LIN {X 0,Y 41.903,Z 386.34,A -85,B 0,C 180,E1 -30757.287,E2 -30757.287} C_VEL
LIN {X 0,Y 51.448,Z 382.345,A -85,B 0,C 180,E1 -30762.982,E2 -30762.982} C_VEL
LIN {X 0,Y 62.953,Z 376.201,A -85,B 0,C 180,E1 -30767.635,E2 -30767.635} C_VEL
LIN {X 0,Y 67.152,Z 373.585,A -85,B 0,C 180,E1 -30768.916,E2 -30768.916} C_VEL
LIN {X 0,Y 68.053,Z 372.62,A -85,B 0,C 180,E1 -30771.442,E2 -30771.442} C_VEL
LIN {X 0,Y 68.483,Z 372.007,A -85,B 0,C 180,E1 -30774.11,E2 -30774.11} C_VEL
LIN {X 0,Y 69.377,Z 371.006,A -85,B 0,C 180,E1 -30780,E2 -30780} C_VEL
LIN {X 0,Y 68.315,Z 371.733,A -85,B 0,C 180,E1 -30786.282,E2 -30786.282} C_VEL
LIN {X 0,Y 67.497,Z 372.745,A -85,B 0,C 180,E1 -30792.02,E2 -30792.02} C_VEL
LIN {X 0,Y 65.091,Z 374.375,A -85,B 0,C 180,E1 -30793.653,E2 -30793.653} C_VEL
LIN {X 0,Y 55.192,Z 379.863,A -85,B 0,C 180,E1 -30797.248,E2 -30797.248} C_VEL
LIN {X 0,Y 45.566,Z 384.168,A -85,B 0,C 180,E1 -30802.27,E2 -30802.27} C_VEL
LIN {X 0,Y 39.483,Z 386.44,A -85,B 0,C 180,E1 -30807.129,E2 -30807.129} C_VEL
LIN {X 0,Y 33.706,Z 388.286,A -85,B 0,C 180,E1 -30813.485,E2 -30813.485} C_VEL
LIN {X 0,Y 24.157,Z 390.65,A -85,B 0,C 180,E1 -30834.42,E2 -30834.42} C_VEL
LIN {X 0,Y 20.214,Z 391.471,A -85,B 0,C 180,E1 -30870.002,E2 -30870.002} C_VEL
LIN {X 0,Y 21.184,Z 391.275,A -85,B 0,C 180,E1 -30889.377,E2 -30889.377} C_VEL
LIN {X 0,Y 24.157,Z 390.689,A -85,B 0,C 180,E1 -30905.583,E2 -30905.583} C_VEL
LIN {X 0,Y 33.7,Z 388.363,A -85,B 0,C 180,E1 -30926.534,E2 -30926.534} C_VEL
LIN {X 0,Y 42.47,Z 385.492,A -85,B 0,C 180,E1 -30935.528,E2 -30935.528} C_VEL
LIN {X 0,Y 51.924,Z 381.593,A -85,B 0,C 180,E1 -30941.348,E2 -30941.348} C_VEL
LIN {X 0,Y 61.757,Z 376.558,A -85,B 0,C 180,E1 -30945.311,E2 -30945.311} C_VEL
LIN {X 0,Y 65.067,Z 374.577,A -85,B 0,C 180,E1 -30946.437,E2 -30946.437} C_VEL
LIN {X 0,Y 67.575,Z 372.915,A -85,B 0,C 180,E1 -30947.994,E2 -30947.994} C_VEL
LIN {X 0,Y 68.471,Z 371.834,A -85,B 0,C 180,E1 -30954.108,E2 -30954.108} C_VEL
LIN {X 0,Y 69.414,Z 371.202,A -85,B 0,C 180,E1 -30960,E2 -30960} C_VEL
LIN {X 0,Y 68.511,Z 372.201,A -85,B 0,C 180,E1 -30965.888,E2 -30965.888} C_VEL
LIN {X 0,Y 68.081,Z 372.809,A -85,B 0,C 180,E1 -30968.536,E2 -30968.536} C_VEL
LIN {X 0,Y 67.185,Z 373.763,A -85,B 0,C 180,E1 -30971.024,E2 -30971.024} C_VEL
LIN {X 0,Y 57.972,Z 379.2,A -85,B 0,C 180,E1 -30974.102,E2 -30974.102} C_VEL
LIN {X 0,Y 48.205,Z 383.911,A -85,B 0,C 180,E1 -30978.615,E2 -30978.615} C_VEL
LIN {X 0,Y 40.64,Z 386.879,A -85,B 0,C 180,E1 -30983.695,E2 -30983.695} C_VEL
LIN {X 0,Y 35.481,Z 388.501,A -85,B 0,C 180,E1 -30987.316,E2 -30987.316} C_VEL
LIN {X 0,Y 26.338,Z 390.564,A -85,B 0,C 180,E1 -30993.352,E2 -30993.352} C_VEL
LIN {X 0,Y 19.232,Z 391.658,A -85,B 0,C 180,E1 -31002.01,E2 -31002.01} C_VEL
LIN {X 0,Y 14.953,Z 392.123,A -85,B 0,C 180,E1 -31015.802,E2 -31015.802} C_VEL
LIN {X 0,Y 14.005,Z 392.204,A -85,B 0,C 180,E1 -31022.658,E2 -31022.658} C_VEL
LIN {X 0,Y 12.922,Z 392.404,A -85,B 0,C 180,E1 -31049.997,E2 -31049.997} C_VEL
LIN {X 0,Y 14.249,Z 392.164,A -85,B 0,C 180,E1 -31079.551,E2 -31079.551} C_VEL
LIN {X 0,Y 23.758,Z 390.517,A -85,B 0,C 180,E1 -31112.55,E2 -31112.55} C_VEL
LIN {X 0,Y 29.881,Z 389.097,A -85,B 0,C 180,E1 -31120.184,E2 -31120.184} C_VEL
LIN {X 0,Y 39.699,Z 386.138,A -85,B 0,C 180,E1 -31126.818,E2 -31126.818} C_VEL
LIN {X 0,Y 49.828,Z 382.143,A -85,B 0,C 180,E1 -31130.859,E2 -31130.859} C_VEL
LIN {X 0,Y 60.081,Z 377.013,A -85,B 0,C 180,E1 -31133.702,E2 -31133.702} C_VEL
LIN {X 0,Y 62.486,Z 375.502,A -85,B 0,C 180,E1 -31135.463,E2 -31135.463} C_VEL
LIN {X 0,Y 63.214,Z 374.832,A -85,B 0,C 180,E1 -31140,E2 -31140} C_VEL
LIN {X 0,Y 62.047,Z 375.53,A -85,B 0,C 180,E1 -31146.504,E2 -31146.504} C_VEL
LIN {X 0,Y 59.578,Z 376.988,A -85,B 0,C 180,E1 -31148.419,E2 -31148.419} C_VEL
LIN {X 0,Y 50.119,Z 381.647,A -85,B 0,C 180,E1 -31151.014,E2 -31151.014} C_VEL
LIN {X 0,Y 40.065,Z 385.585,A -85,B 0,C 180,E1 -31155.255,E2 -31155.255} C_VEL
LIN {X 0,Y 30.365,Z 388.487,A -85,B 0,C 180,E1 -31162.214,E2 -31162.214} C_VEL
LIN {X 0,Y 18.838,Z 390.85,A -85,B 0,C 180,E1 -31181.746,E2 -31181.746} C_VEL
LIN {X 0,Y 14.695,Z 391.451,A -85,B 0,C 180,E1 -31201.43,E2 -31201.43} C_VEL
LIN {X 0,Y 13.126,Z 391.67,A -85,B 0,C 180,E1 -31230.003,E2 -31230.003} C_VEL
LIN {X 0,Y 14.695,Z 391.474,A -85,B 0,C 180,E1 -31258.575,E2 -31258.575} C_VEL
LIN {X 0,Y 18.839,Z 390.888,A -85,B 0,C 180,E1 -31278.259,E2 -31278.259} C_VEL
LIN {X 0,Y 30.361,Z 388.563,A -85,B 0,C 180,E1 -31297.814,E2 -31297.814} C_VEL
LIN {X 0,Y 40.052,Z 385.691,A -85,B 0,C 180,E1 -31304.822,E2 -31304.822} C_VEL
LIN {X 0,Y 50.106,Z 381.792,A -85,B 0,C 180,E1 -31309.068,E2 -31309.068} C_VEL
LIN {X 0,Y 59.607,Z 377.147,A -85,B 0,C 180,E1 -31311.675,E2 -31311.675} C_VEL
LIN {X 0,Y 62.131,Z 375.679,A -85,B 0,C 180,E1 -31313.505,E2 -31313.505} C_VEL
LIN {X 0,Y 63.217,Z 375.024,A -85,B 0,C 180,E1 -31320,E2 -31320} C_VEL
LIN {X 0,Y 62.53,Z 375.663,A -85,B 0,C 180,E1 -31324.467,E2 -31324.467} C_VEL
LIN {X 0,Y 60.073,Z 377.187,A -85,B 0,C 180,E1 -31326.205,E2 -31326.205} C_VEL
LIN {X 0,Y 49.827,Z 382.279,A -85,B 0,C 180,E1 -31329.124,E2 -31329.124} C_VEL
LIN {X 0,Y 37.646,Z 386.903,A -85,B 0,C 180,E1 -31334.277,E2 -31334.277} C_VEL
LIN {X 0,Y 29.883,Z 389.169,A -85,B 0,C 180,E1 -31339.819,E2 -31339.819} C_VEL
LIN {X 0,Y 18.307,Z 391.57,A -85,B 0,C 180,E1 -31359.839,E2 -31359.839} C_VEL
LIN {X 0,Y 14.005,Z 392.204,A -85,B 0,C 180,E1 -31382.658,E2 -31382.658} C_VEL
LIN {X 0,Y 12.565,Z 392.34,A -85,B 0,C 180,E1 -31398.466,E2 -31398.466} C_VEL
LIN {X 0,Y 11.583,Z 392.336,A -85,B 0,C 180,E1 -31416.647,E2 -31416.647} C_VEL
LIN {X 0,Y 12.363,Z 391.94,A -85,B 0,C 180,E1 -31455.277,E2 -31455.277} C_VEL
LIN {X 0,Y 17.093,Z 391.118,A -85,B 0,C 180,E1 -31481.192,E2 -31481.192} C_VEL
LIN {X 0,Y 23.133,Z 390.009,A -85,B 0,C 180,E1 -31490.981,E2 -31490.981} C_VEL
LIN {X 0,Y 24.078,Z 389.762,A -85,B 0,C 180,E1 -31491.657,E2 -31491.657} C_VEL
LIN {X 0,Y 35.215,Z 387.014,A -85,B 0,C 180,E1 -31496.249,E2 -31496.249} C_VEL
LIN {X 0,Y 45.696,Z 383.376,A -85,B 0,C 180,E1 -31498.547,E2 -31498.547} C_VEL
LIN {X 0,Y 56.224,Z 378.626,A -85,B 0,C 180,E1 -31500.155,E2 -31500.155} C_VEL
LIN {X 0,Y 56.254,Z 378.578,A -85,B 0,C 180,E1 -31501.901,E2 -31501.901} C_VEL
LIN {X 0,Y 45.764,Z 383.265,A -85,B 0,C 180,E1 -31503.451,E2 -31503.451} C_VEL
LIN {X 0,Y 35.341,Z 386.842,A -85,B 0,C 180,E1 -31506.129,E2 -31506.129} C_VEL
LIN {X 0,Y 28.448,Z 388.688,A -85,B 0,C 180,E1 -31508.827,E2 -31508.827} C_VEL
LIN {X 0,Y 15.075,Z 391.05,A -85,B 0,C 180,E1 -31521.194,E2 -31521.194} C_VEL
LIN {X 0,Y 9.119,Z 391.651,A -85,B 0,C 180,E1 -31539.592,E2 -31539.592} C_VEL
LIN {X 0,Y 6.027,Z 391.87,A -85,B 0,C 180,E1 -31590.007,E2 -31590.007} C_VEL
LIN {X 0,Y 9.12,Z 391.673,A -85,B 0,C 180,E1 -31640.414,E2 -31640.414} C_VEL
LIN {X 0,Y 15.076,Z 391.088,A -85,B 0,C 180,E1 -31658.811,E2 -31658.811} C_VEL
LIN {X 0,Y 28.447,Z 388.762,A -85,B 0,C 180,E1 -31671.212,E2 -31671.212} C_VEL
LIN {X 0,Y 38.8,Z 385.891,A -85,B 0,C 180,E1 -31675.035,E2 -31675.035} C_VEL
LIN {X 0,Y 49.255,Z 381.991,A -85,B 0,C 180,E1 -31677.22,E2 -31677.22} C_VEL
LIN {X 0,Y 56.253,Z 378.755,A -85,B 0,C 180,E1 -31678.173,E2 -31678.173} C_VEL
LIN {X 0,Y 56.225,Z 378.801,A -85,B 0,C 180,E1 -31679.826,E2 -31679.826} C_VEL
LIN {X 0,Y 45.697,Z 383.513,A -85,B 0,C 180,E1 -31681.447,E2 -31681.447} C_VEL
LIN {X 0,Y 35.216,Z 387.113,A -85,B 0,C 180,E1 -31683.756,E2 -31683.756} C_VEL
LIN {X 0,Y 28.273,Z 388.969,A -85,B 0,C 180,E1 -31686.108,E2 -31686.108} C_VEL
LIN {X 0,Y 14.79,Z 391.37,A -85,B 0,C 180,E1 -31698.118,E2 -31698.118} C_VEL
LIN {X 0,Y 7.974,Z 392.021,A -85,B 0,C 180,E1 -31722.351,E2 -31722.351} C_VEL
LIN {X 0,Y 5.817,Z 392.204,A -85,B 0,C 180,E1 -31769.993,E2 -31769.993} C_VEL
LIN {X 0,Y 8.793,Z 391.963,A -85,B 0,C 180,E1 -31823.054,E2 -31823.054} C_VEL
LIN {X 0,Y 21.424,Z 390.316,A -85,B 0,C 180,E1 -31849.771,E2 -31849.771} C_VEL
LIN {X 0,Y 24.078,Z 389.762,A -85,B 0,C 180,E1 -31851.657,E2 -31851.657} C_VEL
LIN {X 0,Y 26.399,Z 391.723,A -85,B 0,C 180,E1 -31852.986,E2 -31852.986} C_VEL
LIN {X 0,Y 26.399,Z 600,A -85,B 0,C 180,E1 -31852.986,E2 -31852.986} C_VEL
LIN {X 0,Y 26.399,Z 600,A -85,B 0,C 180,E1 -31852.986,E2 -31852.986}

QRS_NEXT_CUT()

QRS_NEXT()
QRS_HOME()

END
